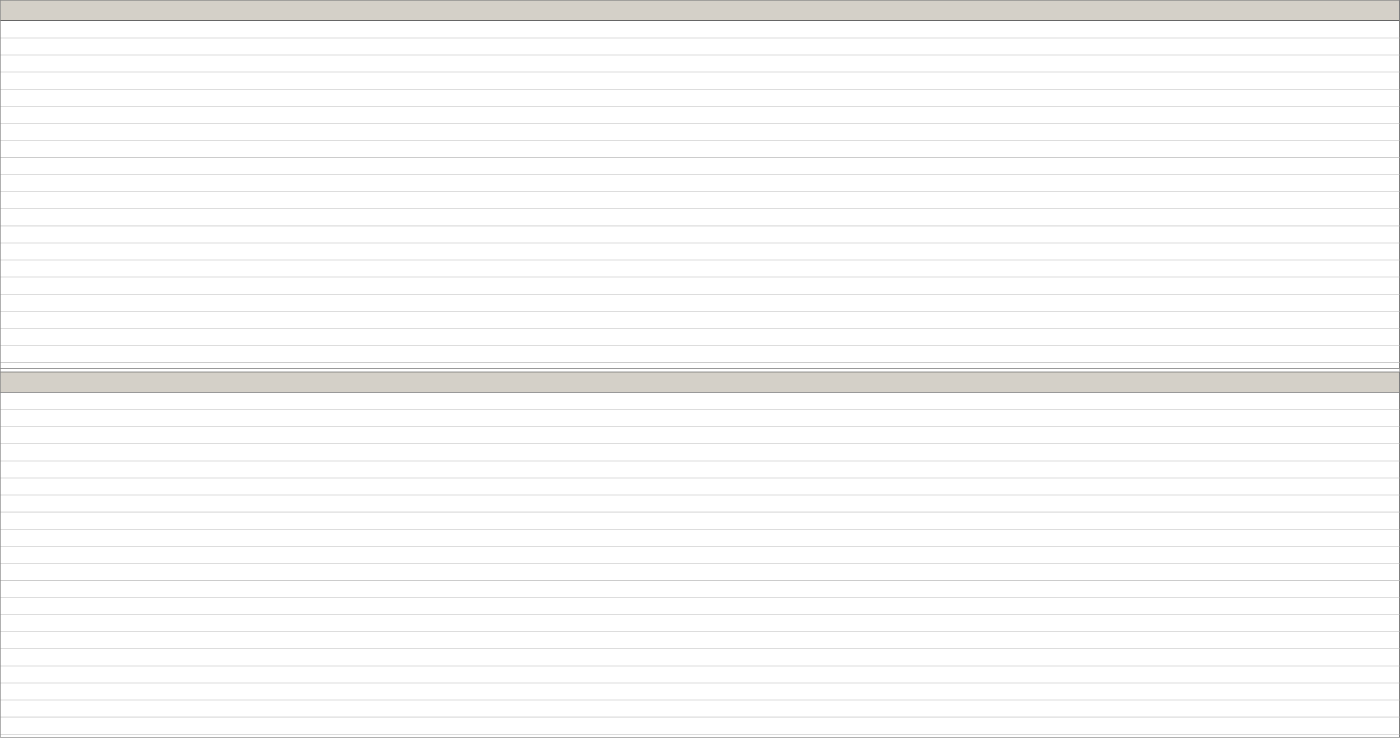
VISUALIZATION v_alarm  // 2048x1080
    Table (0,0 2048x539), data array: GVL.alarms1_hmi
        p3104783080: GVL.fb_buffer.fb_rollers[INDEX].AxisRef
        p2501879983: GVL.fb_buffer.fb_rollers[INDEX].current_tote_status
        p7306298: GVL.fb_buffer.fb_rollers[INDEX].ton_timeout
        p1933151965: GVL.fb_buffer.fb_rollers[INDEX].eStates
        p3863566920: GVL.fb_buffer.fb_rollers[INDEX].iStateTemp
        p2192122294: GVL.fb_buffer.fb_rollers[INDEX].errorMessage
        p400160035: GVL.fb_buffer.fb_rollers[INDEX].xError
        p1265227338: GVL.fb_buffer.fb_rollers[INDEX].rPos_up
        p3726181087: GVL.fb_buffer.fb_rollers[INDEX].rPos_down
        p3854506369: GVL.alarms1_hmi[INDEX].msg
        p1892666644: GVL.alarms1_hmi[INDEX].str_DT
        p338671338: GVL.PackTags.Admin.Alarm[INDEX].Value
        p2170511999: GVL.PackTags.Admin.Alarm[INDEX].Message
        p3723444502: GVL.PackTags.Admin.Alarm[INDEX].Category
        p1218418051: GVL.PackTags.Admin.Alarm[INDEX].DateTime
        p746581629: GVL.PackTags.Admin.Alarm[INDEX].AckDateTime
        p511219082: Datetime
    Table (0,544 2048x535), data array: GVL.alarms2_hmi
        p3104783080: GVL.fb_buffer.fb_rollers[INDEX].AxisRef
        p2501879983: GVL.fb_buffer.fb_rollers[INDEX].current_tote_status
        p7306298: GVL.fb_buffer.fb_rollers[INDEX].ton_timeout
        p1933151965: GVL.fb_buffer.fb_rollers[INDEX].eStates
        p3863566920: GVL.fb_buffer.fb_rollers[INDEX].iStateTemp
        p2192122294: GVL.fb_buffer.fb_rollers[INDEX].errorMessage
        p400160035: GVL.fb_buffer.fb_rollers[INDEX].xError
        p1265227338: GVL.fb_buffer.fb_rollers[INDEX].rPos_up
        p3726181087: GVL.fb_buffer.fb_rollers[INDEX].rPos_down
        p3854506369: GVL.alarms2_hmi[INDEX].msg
        p1892666644: GVL.alarms2_hmi[INDEX].str_DT
        p338671338: GVL.PackTags.Admin.Alarm[INDEX].Value
        p2170511999: GVL.PackTags.Admin.Alarm[INDEX].Message
        p3723444502: GVL.PackTags.Admin.Alarm[INDEX].Category
        p1218418051: GVL.PackTags.Admin.Alarm[INDEX].DateTime
        p746581629: GVL.PackTags.Admin.Alarm[INDEX].AckDateTime
        p511219082: Datetime
END_VISUALIZATION

(* stored: Version 1.1.0.1, ProductVersion 3.1.4024.12
   Visu v_alarm: Id {51d6440c-068c-4c8c-a478-475ae0c9cee1} *)
